// TIA Portal V17 export
// export: Created 2022-06-16T09:21:04.8875112Z, ExportSetting WithDefaults, DisplayName Totally Integrated Automation Portal, DisplayVersion V17, DisplayName TIA Portal Openness, DisplayVersion V17, DisplayName TIA Portal Version Control Interface, DisplayVersion V17, DisplayName STEP 7 Professional, DisplayVersion V17, DisplayName STEP 7 Safety, DisplayVersion V17, DisplayName WinCC Advanced, DisplayVersion V17
FUNCTION "Rapport_Mécanique" : Void   // FC70, LAD
{ S7_Optimized_Access := 'TRUE' }
VERSION : 0.1
// stored: AutoNumber false, IsIECCheckEnabled false, SetENOAutomatically false, UDAEnableTagReadback false
BEGIN

REGION Network 1: Test du bloc CylPos
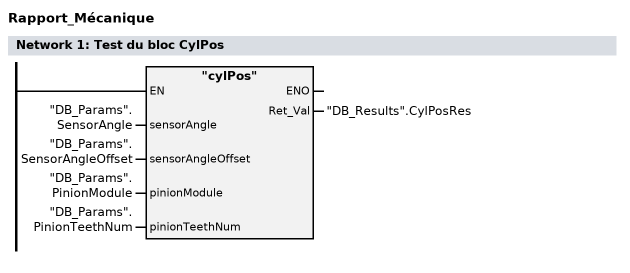
   RUNG wire#powerrail
      "cylPos"(sensorAngle := "DB_Params".SensorAngle, sensorAngleOffset := "DB_Params".SensorAngleOffset, pinionModule := "DB_Params".PinionModule, pinionTeethNum := "DB_Params".PinionTeethNum, Ret_Val => "DB_Results".CylPosRes)
   END_RUNG
   // the same network as SCL:
   "DB_Results".CylPosRes := "cylPos"(sensorAngle := "DB_Params".SensorAngle,
                           sensorAngleOffset := "DB_Params".SensorAngleOffset,
                           pinionModule := "DB_Params".PinionModule,
                           pinionTeethNum := "DB_Params".PinionTeethNum);
END_REGION
END_FUNCTION
